FUNCTION_BLOCK FB_CRYO_THLD_BASE
VAR_INPUT
	in_nMode:		E_CRYO_THLD_MODE := E_CRYO_THLD_MODE.FIXED;
	in_aThld:		ARRAY [1..4] OF LREAL;	// Array of fixed thresholds. See E_CRYO_ALARM_LEVELS and E_CRYO_ALARM_IDX.
	in_aThldDelay:	ARRAY [1..4] OF UDINT;	// Array of delays for each threshold [ms].
	in_lrHyst:		LREAL := 0.0;			// Hysteresis value, percent or absolute (see in_bHystPct)
	in_bHystPct:	BOOL := TRUE;			// If TRUE, hysteresis is in %, otherwise absolute value.
	in_lrValue:		LREAL;					// Value to compare against the thresholds
	in_lrPar1:		LREAL := 0.0;			// Par1, e.g. temperature, for ACTIVE thresholds
END_VAR
VAR_OUTPUT
	out_aThld:			ARRAY [1..4] OF LREAL;	// Active thresholds
	out_nAlarmState:	E_CRYO_ALARM_LEVEL	:= E_CRYO_ALARM_LEVEL.NORMAL;	// Alarm state, e.g. ALARM_HIGH
	out_sAlarmState:	STRING := 'NORMAL';	// Alarm state as a string, e.g. 'ALARM HIGH'
END_VAR
VAR
	timer:	TON;
END_VAR

// Set thresholds
M_SetThresholds();

// Compare input value against the thresholds
M_CheckAlarms();

METHOD M_CheckAlarms : BOOL
VAR_INPUT
END_VAR
VAR
	lrHyst:	LREAL;
END_VAR

// Execute the delay timer.
timer();

//
// Check the input value against the thresholds
// and set alarms and warnings.
// If configured for, activate alarms after a delay.
// Note: the value is compared against the OUT Thresholds !!!
//
CASE out_nAlarmState OF
	E_CRYO_ALARM_LEVEL.NORMAL:
		IF in_lrValue > out_aThld[E_CRYO_ALARM_IDX.ALARM_HIGH] THEN
			IF in_aThldDelay[E_CRYO_ALARM_IDX.ALARM_HIGH] > 0	THEN
				// Activation delay is configured.
				// Start the timer and change state to WARNING_HIGH.
				timer(IN:=FALSE);
				timer(IN:=TRUE, PT:=UDINT_TO_TIME(in_aThldDelay[E_CRYO_ALARM_IDX.ALARM_HIGH]));
				out_nAlarmState	:= E_CRYO_ALARM_LEVEL.WARNING_HIGH;
			ELSE
				timer(IN:=FALSE);
				out_nAlarmState	:= E_CRYO_ALARM_LEVEL.ALARM_HIGH;
			END_IF
		ELSIF in_lrValue < out_aThld[E_CRYO_ALARM_IDX.ALARM_LOW] THEN
			IF in_aThldDelay[E_CRYO_ALARM_IDX.ALARM_LOW] > 0	THEN
				// Activation delay is configured.
				// Start the timer and change state to WARNING_LOW.
				timer(IN:=FALSE);
				timer(IN:=TRUE, PT:=UDINT_TO_TIME(in_aThldDelay[E_CRYO_ALARM_IDX.ALARM_LOW]));
				out_nAlarmState	:= E_CRYO_ALARM_LEVEL.WARNING_LOW;
			ELSE
				timer(IN:=FALSE);
				out_nAlarmState	:= E_CRYO_ALARM_LEVEL.ALARM_LOW;
			END_IF
		ELSIF in_lrValue > out_aThld[E_CRYO_ALARM_IDX.WARNING_HIGH] THEN
			IF in_aThldDelay[E_CRYO_ALARM_IDX.WARNING_HIGH] > 0	THEN
				// Activation delay is configured.
				// Activate the warning once the timer expires.
				timer(IN:=TRUE, PT:=UDINT_TO_TIME(in_aThldDelay[E_CRYO_ALARM_IDX.WARNING_HIGH]));
				IF timer.Q	THEN
					IF in_lrValue > out_aThld[E_CRYO_ALARM_IDX.ALARM_HIGH] THEN
						// It might be that due to the delay the alarm level has been reached.
						out_nAlarmState	:= E_CRYO_ALARM_LEVEL.ALARM_HIGH;
					ELSE
						out_nAlarmState	:= E_CRYO_ALARM_LEVEL.WARNING_HIGH;
					END_IF
				END_IF
			ELSE
				timer(IN:=FALSE);
				out_nAlarmState	:= E_CRYO_ALARM_LEVEL.WARNING_HIGH;
			END_IF
		ELSIF	in_lrValue < out_aThld[E_CRYO_ALARM_IDX.WARNING_LOW]	THEN
			IF in_aThldDelay[E_CRYO_ALARM_IDX.WARNING_LOW] > 0	THEN
				// Activation delay is configured.
				// Activate the warning once the timer expires.
				timer(IN:=TRUE, PT:=UDINT_TO_TIME(in_aThldDelay[E_CRYO_ALARM_IDX.WARNING_LOW]));
				IF timer.Q	THEN
					IF in_lrValue < out_aThld[E_CRYO_ALARM_IDX.ALARM_LOW] THEN
						// It might be that due to the delay the alarm level has been reached.
						out_nAlarmState	:= E_CRYO_ALARM_LEVEL.ALARM_LOW;
					ELSE
						out_nAlarmState	:= E_CRYO_ALARM_LEVEL.WARNING_LOW;
					END_IF
				END_IF
			ELSE
				timer(IN:=FALSE);
				out_nAlarmState	:= E_CRYO_ALARM_LEVEL.WARNING_LOW;
			END_IF
		ELSE
			timer(IN:=FALSE);
		END_IF
	E_CRYO_ALARM_LEVEL.WARNING_HIGH:
		lrHyst	:= M_GetHysteresis(E_CRYO_ALARM_IDX.WARNING_HIGH);
		IF	in_lrValue > out_aThld[E_CRYO_ALARM_IDX.ALARM_HIGH]	THEN
			IF in_aThldDelay[E_CRYO_ALARM_IDX.ALARM_HIGH] > 0	THEN
				// Activation delay is configured.
				// Activate the alarm once the timer expires.
				timer(IN:=TRUE, PT:=UDINT_TO_TIME(in_aThldDelay[E_CRYO_ALARM_IDX.ALARM_HIGH]));
				IF timer.Q	THEN
					out_nAlarmState	:= E_CRYO_ALARM_LEVEL.ALARM_HIGH;
				END_IF
			ELSE
				timer(IN:=FALSE);
				out_nAlarmState	:= E_CRYO_ALARM_LEVEL.ALARM_HIGH;
			END_IF
		ELSIF in_lrValue < (out_aThld[E_CRYO_ALARM_IDX.WARNING_HIGH] - lrHyst) THEN
			timer(IN:=FALSE);
			out_nAlarmState	:= E_CRYO_ALARM_LEVEL.NORMAL;
		ELSE
			timer(IN:=FALSE);
		END_IF
	E_CRYO_ALARM_LEVEL.WARNING_LOW:
		lrHyst	:= M_GetHysteresis(E_CRYO_ALARM_IDX.WARNING_LOW);
		IF	in_lrValue < out_aThld[E_CRYO_ALARM_IDX.ALARM_LOW]	THEN
			IF in_aThldDelay[E_CRYO_ALARM_IDX.ALARM_LOW] > 0	THEN
				// Activation delay is configured.
				// Activate the alarm once the timer expires.
				timer(IN:=TRUE, PT:=UDINT_TO_TIME(in_aThldDelay[E_CRYO_ALARM_IDX.ALARM_LOW]));
				IF timer.Q	THEN
					out_nAlarmState	:= E_CRYO_ALARM_LEVEL.ALARM_LOW;
				END_IF
			ELSE
				timer(IN:=FALSE);
				out_nAlarmState	:= E_CRYO_ALARM_LEVEL.ALARM_LOW;
			END_IF
		ELSIF in_lrValue > (out_aThld[E_CRYO_ALARM_IDX.WARNING_LOW] + lrHyst) THEN
			timer(IN:=FALSE);
			out_nAlarmState	:= E_CRYO_ALARM_LEVEL.NORMAL;
		ELSE
			timer(IN:=FALSE);
		END_IF
	E_CRYO_ALARM_LEVEL.ALARM_HIGH:
		lrHyst	:= M_GetHysteresis(E_CRYO_ALARM_IDX.ALARM_HIGH);
		IF in_lrValue < (out_aThld[E_CRYO_ALARM_IDX.ALARM_HIGH] - lrHyst) THEN
			out_nAlarmState	:= E_CRYO_ALARM_LEVEL.WARNING_HIGH;
		END_IF
	E_CRYO_ALARM_LEVEL.ALARM_LOW:
		lrHyst	:= M_GetHysteresis(E_CRYO_ALARM_IDX.ALARM_LOW);
		IF in_lrValue > (out_aThld[E_CRYO_ALARM_IDX.ALARM_LOW] + lrHyst) THEN
			out_nAlarmState	:= E_CRYO_ALARM_LEVEL.WARNING_LOW;
		END_IF
END_CASE

// Set alarm level labels
M_UserSetLabel(out_nAlarmState);
END_METHOD

METHOD M_GetHysteresis : LREAL
VAR_INPUT
	in_nIndex:	E_CRYO_ALARM_IDX;
END_VAR
VAR
	lrHyst:	LREAL;
END_VAR
//
// Get the absolute value of hysteresis.
// 
IF in_bHystPct THEN
	// The vaue is given as percentage of threshold.
	lrHyst	:= in_aThld[in_nIndex] * in_lrHyst / 100.0;
ELSE
	// The vaue is given as absolute value.
	lrHyst	:= in_lrHyst;
END_IF

M_GetHysteresis	:= ABS(lrHyst);
END_METHOD

METHOD M_SetThresholds : BOOL
VAR_INPUT
END_VAR
VAR
	i:	INT;
END_VAR
CASE in_nMode OF
	E_CRYO_THLD_MODE.FIXED:
		// Take the input array for thresholds
		FOR i:=1 TO 4 DO
			out_aThld[i]	:= in_aThld[i];
		END_FOR
	E_CRYO_THLD_MODE.ACTIVE:
		// Dynamically set thresholds
		M_UserSetActiveThresholds();
	E_CRYO_THLD_MODE.LAST_ACTIVE:
		// Keep last thresholds. Don't do anything.
		;
END_CASE
END_METHOD

METHOD M_UserSetActiveThresholds : BOOL
// This is a Dummy implementation of active thresholds.
// TODO User: Define specific implementation.
VAR_INPUT
END_VAR
VAR
	i:	INT;
END_VAR
// TODO User
// Define specific implementation.
// This is just an example.
//
out_aThld[E_CRYO_ALARM_IDX.ALARM_LOW]	:= in_aThld[E_CRYO_ALARM_IDX.ALARM_LOW]    + in_lrPar1;
out_aThld[E_CRYO_ALARM_IDX.WARNING_LOW]	:= in_aThld[E_CRYO_ALARM_IDX.WARNING_LOW]  + in_lrPar1;
out_aThld[E_CRYO_ALARM_IDX.WARNING_HIGH]	:= in_aThld[E_CRYO_ALARM_IDX.WARNING_HIGH] - in_lrPar1;
out_aThld[E_CRYO_ALARM_IDX.ALARM_HIGH]	:= in_aThld[E_CRYO_ALARM_IDX.ALARM_HIGH]   - in_lrPar1;
END_METHOD

METHOD M_UserSetLabel : BOOL
VAR_INPUT
	in_nLevel:	E_CRYO_ALARM_LEVEL;
END_VAR
//
// Set labels depending on the alarm level.
// This is the default implementation.
// To be overwritten by User if different labels are needed.
//
CASE in_nLevel OF
	E_CRYO_ALARM_LEVEL.ALARM_LOW:
		out_sAlarmState	:= 'ALARM LOW';
	E_CRYO_ALARM_LEVEL.WARNING_LOW:
		out_sAlarmState	:= 'WARNING LOW';
	E_CRYO_ALARM_LEVEL.NORMAL:
		out_sAlarmState	:= 'NORMAL';
	E_CRYO_ALARM_LEVEL.WARNING_HIGH:
		out_sAlarmState	:= 'WARNING HIGH';
	E_CRYO_ALARM_LEVEL.ALARM_HIGH:
		out_sAlarmState	:= 'ALARM HIGH';
END_CASE
END_METHOD

END_FUNCTION_BLOCK

(* stored: Version 1.1.0.1, ProductVersion 3.1.4024.9
   POU FB_CRYO_THLD_BASE: Id {444425cb-ac17-43d2-88ff-ed23623aa366}, SpecialFunc None
   Method M_CheckAlarms: Id {fd6d363d-95cf-421c-9888-bf474639abc3}
   Method M_GetHysteresis: Id {a1c163dc-0c4c-44fd-9369-2012badcc023}
   Method M_SetThresholds: Id {a93233dd-9155-4b13-bc45-3914752de314}
   Method M_UserSetActiveThresholds: Id {f8fcbf4a-3da3-480e-b5e4-e005cec0e4ff}
   Method M_UserSetLabel: Id {bf781e12-91ec-4d3c-884b-b49bf551b4aa} *)
